// TIA Portal V18 export
FUNCTION "块_1" : Void   // FC1, LAD
{ S7_Optimized_Access := 'TRUE' }
// stored: SetENOAutomatically false
BEGIN

REGION Network 2 (SCL)
   "CheckPositioningOrder_IDB"("V90Servo[3]":="ServoV90_DeviceCtl".V90Servo[3],
                               HaveAxisStart=>"DATA".HaveAxisStart,
                               AxisStartNumber=>"DATA".AxisStartNumber);

   //When the 382A1 card is stuck at step 130, change the process step to 100 and locate it again.
   //当382A1卡在 130步时,修改流程步去100再次定位
   IF    "DATA"."Forced modification"    AND
       "DATA".HaveAxisStart AND "DATA".AxisStartNumber <> 32767 AND
       "V90Servo_DB".Servo_382A1.sStep[1] = 130AND
       "V90Servo_DB".Servo_382A1.sErrorCode=0  AND
      // "ServoV90_A3".Auto.Pos["ServoV90_A3".Auto.Index].Pos<> "ServoV90_A3".Out.oActPosition
       "ServoV90_A3".Auto.Pos[6].Pos<> "ServoV90_A3".Out.oActPosition
   THEN
       "V90Servo_DB".Servo_382A1.sStep[1] := 100
       ;
   END_IF;
END_REGION
END_FUNCTION
